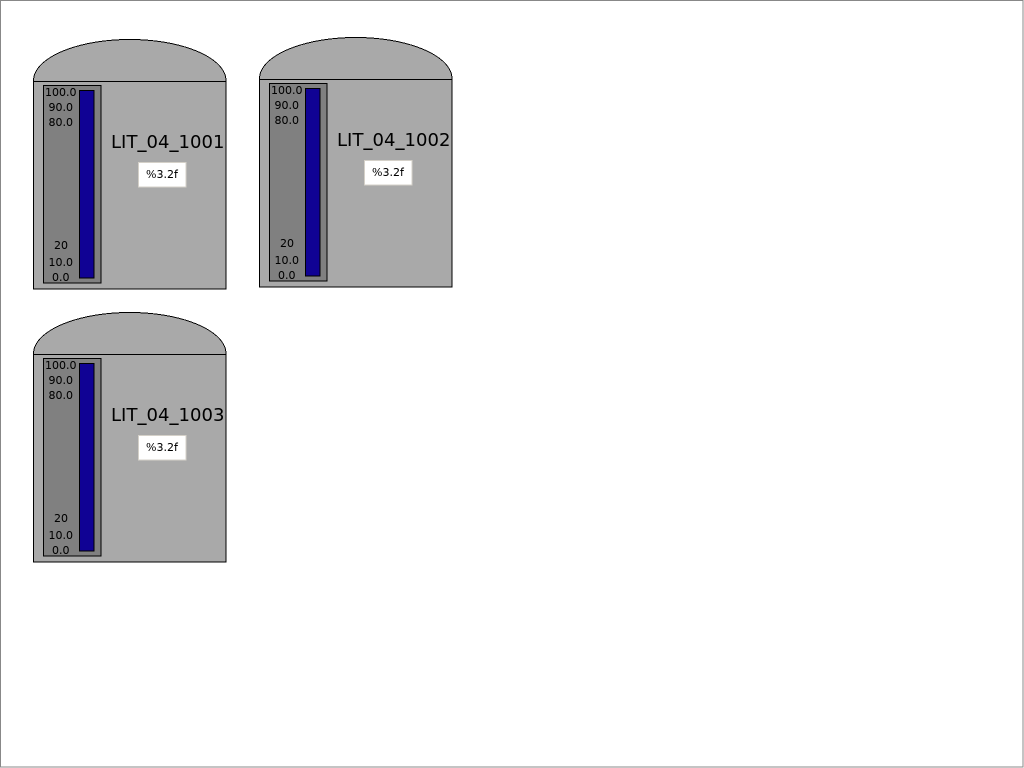
VISUALIZATION Vessel  // 1024x768
    Group (33,39 200x250)
        Ellipse (0,0 193x83)
        Rectangle (0,42 193x208)
        Rectangle (10,46 58x198)
        Rectangle (46,51 15x188)
        Label (10,231 36x15), "0.0"
        Label (10,46 36x15), "100.0"
        Label (10,61 36x15), "90.0"
        Label (10,76 36x15), "80.0"
        Label (10,216 36x15), "10.0"
        Label (10,199 36x15), "20"
        Label (70,88 130x30), "LIT_04_1001"
        Textfield (105,123 48x25), "%3.2f", text variable: progLITCntrl.LIT_04_1001.Level
            OnMouseClick: write progLITCntrl.LIT_04_1001.Level via VisuDialogs.NumpadExtended, min 0.0, max 100.0
    Group (259,37 200x250)
        Ellipse (0,0 193x83)
        Rectangle (0,42 193x208)
        Rectangle (10,46 58x198)
        Rectangle (46,51 15x188)
        Label (10,231 36x15), "0.0"
        Label (10,46 36x15), "100.0"
        Label (10,61 36x15), "90.0"
        Label (10,76 36x15), "80.0"
        Label (10,216 36x15), "10.0"
        Label (10,199 36x15), "20"
        Label (70,88 130x30), "LIT_04_1002"
        Textfield (105,123 48x25), "%3.2f", text variable: progLITCntrl.LIT_04_1002.Level
            OnMouseClick: write progLITCntrl.LIT_04_1002.Level via VisuDialogs.NumpadExtended, min 0.0, max 100.0
    Group (33,312 200x250)
        Ellipse (0,0 193x83)
        Rectangle (0,42 193x208)
        Rectangle (10,46 58x198)
        Rectangle (46,51 15x188)
        Label (10,231 36x15), "0.0"
        Label (10,46 36x15), "100.0"
        Label (10,61 36x15), "90.0"
        Label (10,76 36x15), "80.0"
        Label (10,216 36x15), "10.0"
        Label (10,199 36x15), "20"
        Label (70,88 130x30), "LIT_04_1003"
        Textfield (105,123 48x25), "%3.2f", text variable: progLITCntrl.LIT_04_1003.Level
            OnMouseClick: write progLITCntrl.LIT_04_1003.Level via VisuDialogs.NumpadExtended, min 0.0, max 100.0
END_VISUALIZATION

(* stored: Version 1.1.0.1, ProductVersion 3.1.4022.17
   Visu Vessel: Id {ceffee4c-a57c-4651-a662-50df9badb628} *)
